FUNCTION_BLOCK FB_RotateStation EXTENDS FB_XPlanarStationBase
VAR
	_StationAngle  : LREAL;
	_NumberOfTurns : DINT;
END_VAR

METHOD Execute
VAR_INST
	i			  : UDINT := 1;
	CommandResult : I_PlanarTaskResult;
END_VAR
SUPER^.Execute();
IF StationState = E_XPlanarStationState.ProcessMover THEN
	CommandResult := ipCurrentMover.MoveCommand.Rotate(_StationAngle, _NumberOfTurns);
	IF CommandResult.Done THEN
		_StationComplete := TRUE;
	ELSIF CommandResult.Error THEN
		; //Command returned an error!
	END_IF
END_IF
END_METHOD

PROPERTY NumberOfTurns : DINT
SET
_NumberOfTurns := NumberOfTurns;
END_SET
END_PROPERTY

PROPERTY StationAngle : LREAL
SET
_StationAngle := StationAngle;
END_SET
END_PROPERTY

END_FUNCTION_BLOCK

(* stored: Version 1.1.0.1, ProductVersion 3.1.4024.13
   POU FB_RotateStation: Id {d0ee9b9c-eeff-4082-9db1-0bc32eab28c5}, SpecialFunc None
   Method Execute: Id {2be4b8cf-b65d-43e3-92eb-e6a95a99401e}
   Property NumberOfTurns: Id {9d661a2e-f7f3-4558-afb3-350c215cc0c4}
   Set Set: Id {cad60f88-e9df-4e9a-94e5-e7e43cc8e24a}
   Property StationAngle: Id {568cd894-6b94-4015-b665-4e2c3332f5de}
   Set Set: Id {8b016c78-79fe-4d2f-b17c-5ed06ac7ec95} *)
